	DATA_BLOCK DB401
	TITLE =DBG301M  LOUVER HEATING GLASS TUBE HEAT EXCHANGER
	//COPYRIGHT:    (C) 2009  BUHLER AG, CH-9240 UZWIL, SWITZERLAND
	//
	//PRODUCT:      WinCoS_BIW01_09
	//
	//TITLE:        LOUVER HEATING GLASS TUBE HEAT EXCHANGER
	//                Machine group DB
	//                Maschinengruppen-DB
	//
	//-------------------------------------------------------------------------
	//
	//IDENT:        AUTHOR:             DEPT:             DATE:
	//
	//P01_DB401.1.0 K.Renz              CSB41             13.Jan.2010
	//              1st Release
	//
	//-------------------------------------------------------------------------
	//
	//PURPOSE:
	//
	//MANUAL :
	//
	//RESTRICTIONS:
	//
	//-------------------------------------------------------------------------
	AUTHOR  : KR
	FAMILY  : USW
	NAME    : DBG301M
	VERSION : 00.00

	FB401
	BEGIN
	      #Gr.Par.ParObjectNo 	:=30100;
	      #Gr.Par.ParIdling      	:=2;
	      #Gr.Par.ParMgr	        :=True;
	      #Gr.Par.ParWgr	        :=False;
	      #Gr.Par.ParGgr	        :=False;
	      #Gr.Par.ParEmptyingTime 	:=0;
	      #Gr.Par.ParHornCode       :=11;
	//Parameter =A-3258-MXZ11 : LOUVER HEATING GLASS TUBE HEAT EXCHANGER
	      #A_3258_MXZ11.Par.ParObjectNo                             :=30101;
	      #A_3258_MXZ11.Par.ParMsgType                              :=7081;
	      #A_3258_MXZ11.Par.ParHornCode                             :=11;
	      #A_3258_MXZ11.Par.ParMonTime                              :=200;
	      #A_3258_MXZ11.Par.ParPulseTimeHN                          :=0;
	      #A_3258_MXZ11.Par.ParPulseTimeLN                          :=0;
	      #A_3258_MXZ11.Par.ParIdlingTime                           :=0;
	      #A_3258_MXZ11.Par.ParDelayTime                            :=10;
	      #A_3258_MXZ11.Par.ParLogOff                               :=False;
	      #A_3258_MXZ11.Par.ParManual                               :=True;
	      #A_3258_MXZ11.Par.ParPulseValve                           :=True;
	      #A_3258_MXZ11.Par.ParContValve                            :=False;
	      #A_3258_MXZ11.Par.ParManualFlap                           :=False;
	//
	//
	//Parameter =A-3259-MXZ11 : LOUVER HEATING GLASS TUBE HEAT EXCHANGER
	      #A_3259_MXZ11.Par.ParObjectNo                             :=30102;
	      #A_3259_MXZ11.Par.ParMsgType                              :=7081;
	      #A_3259_MXZ11.Par.ParHornCode                             :=11;
	      #A_3259_MXZ11.Par.ParMonTime                              :=200;
	      #A_3259_MXZ11.Par.ParPulseTimeHN                          :=0;
	      #A_3259_MXZ11.Par.ParPulseTimeLN                          :=0;
	      #A_3259_MXZ11.Par.ParIdlingTime                           :=0;
	      #A_3259_MXZ11.Par.ParDelayTime                            :=10;
	      #A_3259_MXZ11.Par.ParLogOff                               :=False;
	      #A_3259_MXZ11.Par.ParManual                               :=True;
	      #A_3259_MXZ11.Par.ParPulseValve                           :=True;
	      #A_3259_MXZ11.Par.ParContValve                            :=False;
	      #A_3259_MXZ11.Par.ParManualFlap                           :=False;
	//
	//
	END_DATA_BLOCK
